// SIMATIC S7-200 project (STEP 7-Micro/WIN), CPU 221 REL 01.10

ORGANIZATION_BLOCK MAIN:OB1
TITLE=PROGRAM COMMENTS
BEGIN
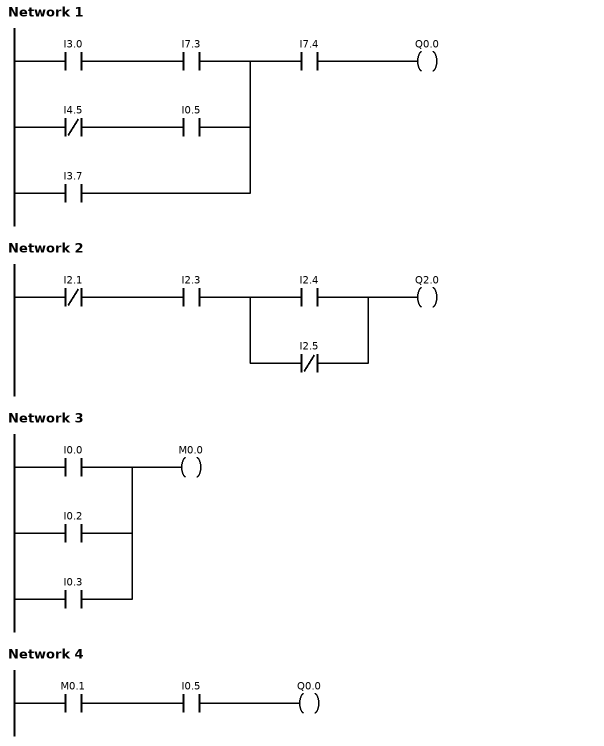
Network 1
LD     I3.0
A      I7.3
LDN    I4.5
A      I0.5
OLD
O      I3.7
A      I7.4
=      Q0.0
Network 2
LDN    I2.1
A      I2.3
LD     I2.4
ON     I2.5
ALD
=      Q2.0
Network 3
LD     I0.0
O      I0.2
O      I0.3
=      M0.0
Network 4
LD     M0.1
A      I0.5
=      Q0.0
END_ORGANIZATION_BLOCK
